{attribute 'signature_flag' := '1073741824'}
FUNCTION_BLOCK PUBLIC JsonParser
VAR_INPUT
	Execute : BOOL; //Parser runs on rising edge of this flag 
	File : STRING(255) := 'C:\Temp\my.json'; //Target json file
	ParseMethod : STRING(255) := 'Read'; //Allowed values are: Read, Write.
	Content : STRING(255); //Variable path
	Port : UINT := 0; //Ads Port for connection. Leave 0 for Port number 851
END_VAR
VAR_OUTPUT
	HasError : BOOL;
	ErrorId : UDINT; //see  ADS error number (https://infosys.beckhoff.com/content/1033/tcplclib_tc2_utilities/45035996647981963.html) or the Win32 error code (https://infosys.beckhoff.com/content/1033/tcplclib_tc2_utilities/27021598155389323.html)
END_VAR
VAR
	startProcess : NT_StartProcess;
	getLocalAmsNetId : FB_GetLocalAmsNetId;
	netIdRead : f_trig;
	initialized : BOOL;
	formatter : FB_FormatString;
END_VAR

startProcess();
getLocalAmsNetId();
startProcess.NETID := getLocalAmsNetId.AddrString;
startProcess.PATHSTR := 'C:\TwinCAT\Functions\Unofficial\JsonReadWriter\TFU003.exe';
startProcess.DIRNAME := 'C:\TwinCAT\Functions\Unofficial\JsonReadWriter\';
formatter(sFormat:='"%s" "%s" "%s"', arg1:=f_string(File), arg2:=f_string(ParseMethod), arg3:=f_string(Content));
IF port <> 0 THEN
	startProcess.COMNDLINE := CONCAT(CONCAT('-AdsPort ',CONCAT(UINT_TO_STRING(Port),' ')),formatter.sOut);
ELSE
	startProcess.COMNDLINE := formatter.sOut;
END_IF

netIdRead(CLK:=getLocalAmsNetId.bBusy, Q=>);

IF netIdRead.Q THEN
	IF NOT getLocalAmsNetId.bError THEN
		initialized := TRUE;
		getLocalAmsNetId.bExecute := FALSE;
	ELSE
		HasError := getLocalAmsNetId.bError;
		ErrorId := getLocalAmsNetId.nErrId;
	END_IF
END_IF

IF NOT initialized THEN
	getLocalAmsNetId.bExecute := TRUE;
END_IF

startProcess.START := initialized AND Execute;

IF initialized THEN
	HasError := startProcess.ERR;
	ErrorId := startProcess.ERRID;
END_IF

END_FUNCTION_BLOCK

(* stored: Version 1.1.0.1, ProductVersion 3.1.4024.3
   POU JsonParser: Id {34d9c780-99db-49b3-b63f-ca9c5a975f9d}, SpecialFunc None *)
